// Mitsubishi GX Works2 project: 0709   PLC: Q02/Q02H

PROGRAM clkCUD
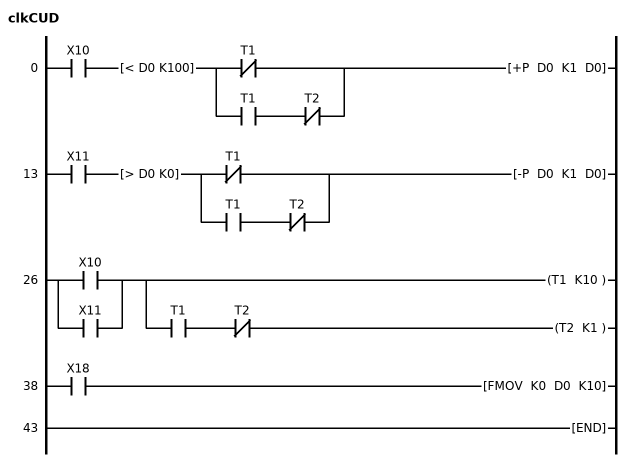
0     LD      X10
      AND<    D0 K100
      LDI     T1
      LD      T1
      ANI     T2
      ORB
      ANB
      +P      D0 K1 D0
13    LD      X11
      AND>    D0 K0
      LDI     T1
      LD      T1
      ANI     T2
      ORB
      ANB
      -P      D0 K1 D0
26    LD      X10
      OR      X11
      OUT     T1 K10
      AND     T1
      ANI     T2
      OUT     T2 K1
38    LD      X18
      FMOV    K0 D0 K10
43    END
END_PROGRAM

PROGRAM DIF_TIME
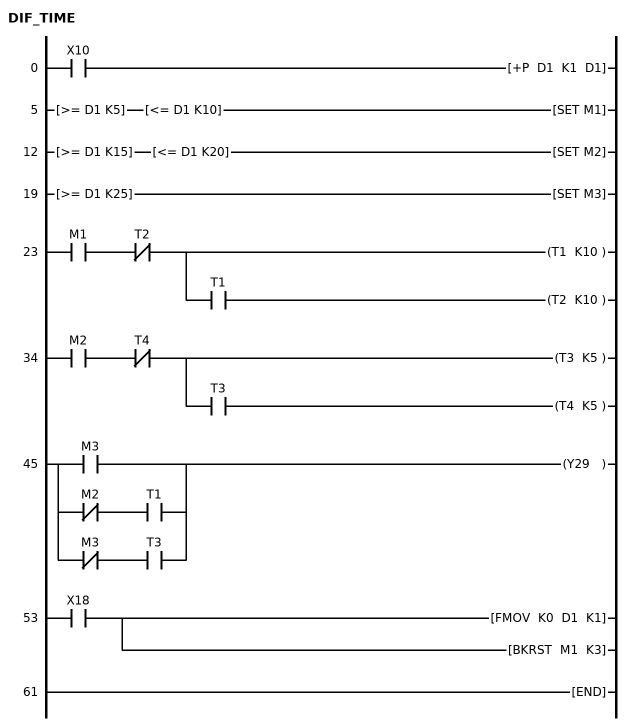
0     LD      X10
      +P      D1 K1 D1
5     LD>=    D1 K5
      AND<=   D1 K10
      SET     M1
12    LD>=    D1 K15
      AND<=   D1 K20
      SET     M2
19    LD>=    D1 K25
      SET     M3
23    LD      M1
      ANI     T2
      OUT     T1 K10
      AND     T1
      OUT     T2 K10
34    LD      M2
      ANI     T4
      OUT     T3 K5
      AND     T3
      OUT     T4 K5
45    LD      M3
      LDI     M2
      AND     T1
      ORB
      LDI     M3
      AND     T3
      ORB
      OUT     Y29
53    LD      X18
      FMOV    K0 D1 K1
      BKRST   M1 K3
61    END
END_PROGRAM

PROGRAM CALC
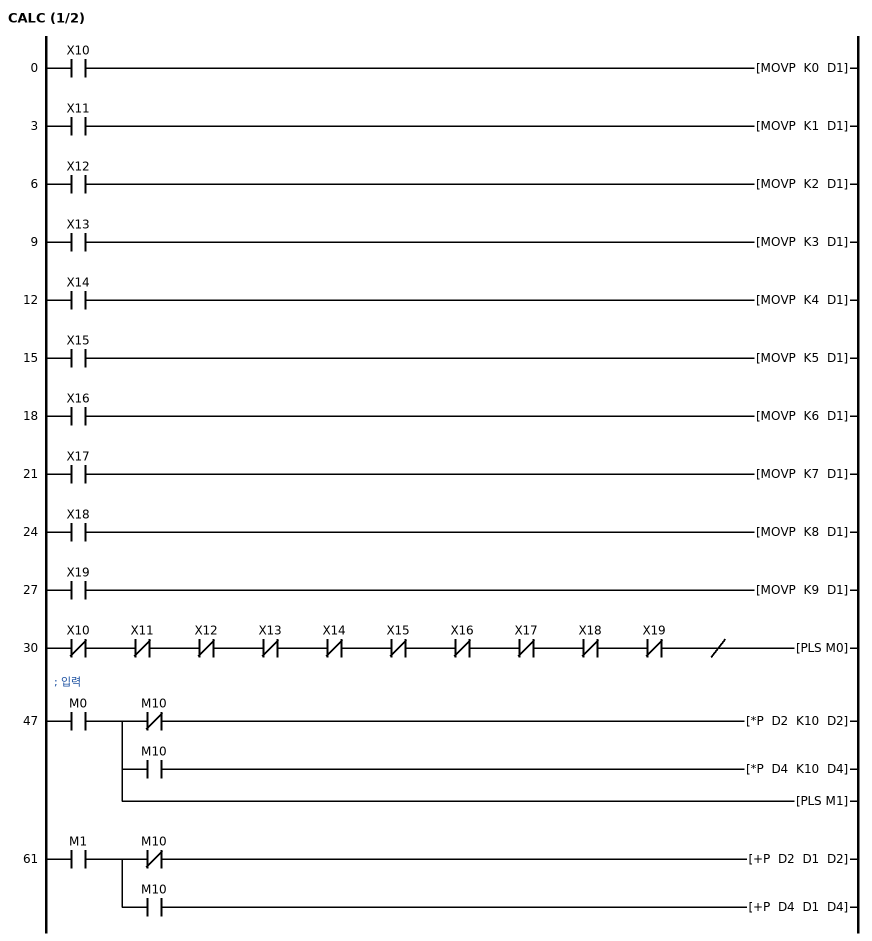
0     LD      X10
      MOVP    K0 D1
3     LD      X11
      MOVP    K1 D1
6     LD      X12
      MOVP    K2 D1
9     LD      X13
      MOVP    K3 D1
12    LD      X14
      MOVP    K4 D1
15    LD      X15
      MOVP    K5 D1
18    LD      X16
      MOVP    K6 D1
21    LD      X17
      MOVP    K7 D1
24    LD      X18
      MOVP    K8 D1
27    LD      X19
      MOVP    K9 D1
30    LDI     X10
      ANI     X11
      ANI     X12
      ANI     X13
      ANI     X14
      ANI     X15
      ANI     X16
      ANI     X17
      ANI     X18
      ANI     X19
      INV
      PLS     M0
; 입력
47    LD      M0
      MPS
      ANI     M10
      *P      D2 K10 D2
      MRD
      AND     M10
      *P      D4 K10 D4
      MPP
      PLS     M1
61    LD      M1
      MPS
      ANI     M10
      +P      D2 D1 D2
      MPP
      AND     M10
      +P      D4 D1 D4
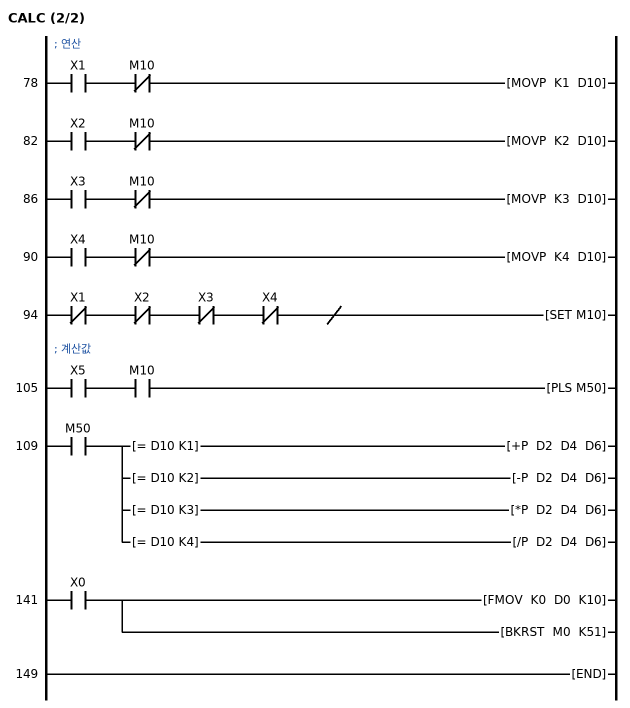
; 연산
78    LD      X1
      ANI     M10
      MOVP    K1 D10
82    LD      X2
      ANI     M10
      MOVP    K2 D10
86    LD      X3
      ANI     M10
      MOVP    K3 D10
90    LD      X4
      ANI     M10
      MOVP    K4 D10
94    LDI     X1
      ANI     X2
      ANI     X3
      ANI     X4
      INV
      SET     M10
; 계산값
105   LD      X5
      AND     M10
      PLS     M50
109   LD      M50
      MPS
      AND=    D10 K1
      +P      D2 D4 D6
      MRD
      AND=    D10 K2
      -P      D2 D4 D6
      MRD
      AND=    D10 K3
      *P      D2 D4 D6
      MPP
      AND=    D10 K4
      /P      D2 D4 D6
141   LD      X0
      FMOV    K0 D0 K10
      BKRST   M0 K51
149   END
END_PROGRAM

PROGRAM txt_calc
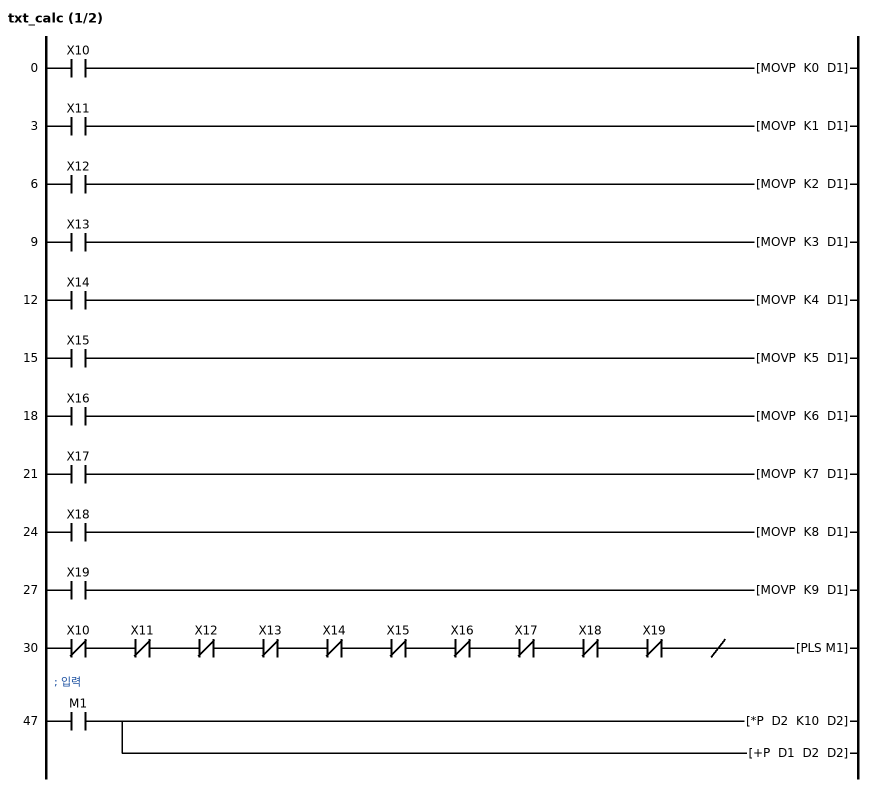
0     LD      X10
      MOVP    K0 D1
3     LD      X11
      MOVP    K1 D1
6     LD      X12
      MOVP    K2 D1
9     LD      X13
      MOVP    K3 D1
12    LD      X14
      MOVP    K4 D1
15    LD      X15
      MOVP    K5 D1
18    LD      X16
      MOVP    K6 D1
21    LD      X17
      MOVP    K7 D1
24    LD      X18
      MOVP    K8 D1
27    LD      X19
      MOVP    K9 D1
30    LDI     X10
      ANI     X11
      ANI     X12
      ANI     X13
      ANI     X14
      ANI     X15
      ANI     X16
      ANI     X17
      ANI     X18
      ANI     X19
      INV
      PLS     M1
; 입력
47    LD      M1
      *P      D2 K10 D2
      +P      D1 D2 D2
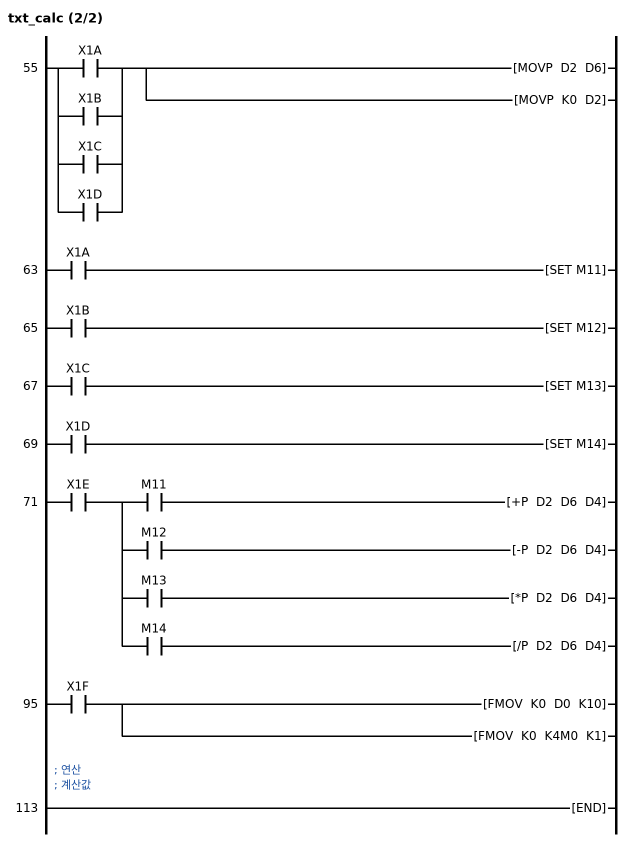
55    LD      X1A
      OR      X1B
      OR      X1C
      OR      X1D
      MOVP    D2 D6
      MOVP    K0 D2
63    LD      X1A
      SET     M11
65    LD      X1B
      SET     M12
67    LD      X1C
      SET     M13
69    LD      X1D
      SET     M14
71    LD      X1E
      MPS
      AND     M11
      +P      D2 D6 D4
      MRD
      AND     M12
      -P      D2 D6 D4
      MRD
      AND     M13
      *P      D2 D6 D4
      MPP
      AND     M14
      /P      D2 D6 D4
95    LD      X1F
      FMOV    K0 D0 K10
      FMOV    K0 K4M0 K1
; 연산
; 계산값
113   END
END_PROGRAM
